FUNCTION_BLOCK IntegrationTestSuite
VAR
	Enable: BOOL;
	MOVETO: BOOL;
	MOVETWO: BOOL;
	DISABLE: BOOL;
	SETBUFFER: BOOL;
END_VAR

// IF Enable THEN
// 	IF succeeded( TestAxis.EnableAxis()) THEN
// 		Enable := FALSE;
// 	END_IF
// END_IF
// 
// IF MOVETO THEN
// 	IF SUCCEEDED(TestAxis.MoveToPosition(1000.0,100.0)) THEN
// 		MOVETO := FALSE;
// 	END_IF
// END_IF
// 
// IF SETBUFFER THEN
// 	SETBUFFER := FALSE;
// 	TestAxis.BufferMode := MC_BufferMode.MC_BlendingLow;
// 	
// END_IF
// 
// IF MOVETWO THEN
// 	IF SUCCEEDED(TestAxis.MoveToPosition(1200.0,200.0)) THEN
// 		MOVETWO := FALSE;
// 	END_IF
// END_IF
// 
// IF DISABLE THEN
// 	IF SUCCEEDED(TestAxis.DisableAxis()) THEN
// 		DISABLE := FALSE;
// 	END_IF
// END_IF
// 
// TestAxis.Cycle();

END_FUNCTION_BLOCK

(* stored: Version 1.1.0.1
   POU IntegrationTestSuite: Id {69bc61fe-8999-4914-8ef6-bb0c95ff7655}, SpecialFunc None *)
